PROGRAM registradorLog21
VAR
	i: INT;
	j: INT;
	k: INT;
END_VAR


IF gvl.logRegister21 <> '' THEN
	FOR i:=100 TO 1 BY -1 DO
		IF gvl_p.arrLogEstufa21[i] <> '' THEN
			gvl_p.arrLogEstufa21[i+1]:= gvl_p.arrLogEstufa21[i];
			gvl_p.arrLogEstufa21[i]:= '';
		END_IF
	END_FOR
	gvl_p.arrLogEstufa21[1]:= concat(gvl_p.arrLogEstufa21[1],gvl.sSystemDateTime);
	gvl_p.arrLogEstufa21[1]:= concat(gvl_p.arrLogEstufa21[1],'    ');
	gvl_p.arrLogEstufa21[1]:= concat(gvl_p.arrLogEstufa21[1],gvl.logRegister21);
	gvl.sCmdInsertLog:= 'INSERT INTO [dbo].[LogGeneral] ([HistoricalTime],[Description])VALUES($'$',$'$')';
	gvl.sCmdInsertLog:= insert(gvl.sCmdInsertLog,gvl.logRegister21,74);	
	gvl.sCmdInsertLog:= insert(gvl.sCmdInsertLog,gvl.sSystemDateTime,71);
	gvl.bInsertLog:=true;
	gvl.logRegister21:= '';
	
	
END_IF

END_PROGRAM

(* stored: Version 1.1.0.1, ProductVersion 3.1.4024.12
   POU registradorLog21: Id {a3f738d1-ef18-4aff-ace1-0dd9de07ce4c}, SpecialFunc None *)
